Staubli VAL3: decodeJointData.pgx

public program decodeJointData(num& x_nStatus (dimensions=1), num& x_nJointData[] (dimensions=1), num& x_nDWordBody[] (dimensions=2), num x_nRowIndex (dimensions=1))
  local num i
begin
  if x_nStatus<0
    return
  endIf
  x_nStatus=0
  for i=0 to size(x_nJointData)-1
    call decodeShareReal(x_nStatus,x_nJointData[i],x_nDWordBody,x_nRowIndex+i)
    if x_nStatus<0
      putln("Failed to decode joint data at index: "+toString("",x_nRowIndex+i))
      return
    endIf
  endFor
end
